TYPE dt_params :
STRUCT
	scale	: LREAL;
	offset	: LREAL;
	f		: WORD;
END_STRUCT
END_TYPE

(* stored: Version 1.1.0.1, ProductVersion 3.1.4024.15
   DUT dt_params: Id {d41c23ff-9e62-4261-bdf7-d75f3d0c1b3e} *)
